TYPE TcoLoggerBuffer :
STRUCT
	Buffer : ARRAY[0..1000] OF TcoMessage;
END_STRUCT
END_TYPE

(* stored: Version 1.1.0.1, ProductVersion 3.1.4024.9
   DUT TcoLoggerBuffer: Id {687c17bc-1ec8-011c-3da7-a90bed9caed3} *)
